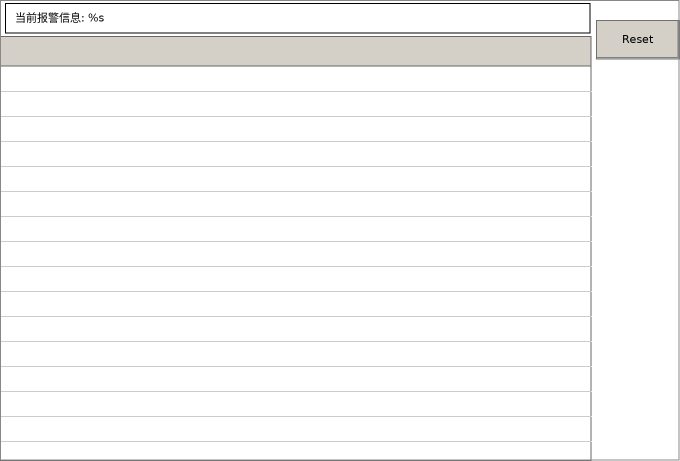
VISUALIZATION Visualization_ActEvent  // 680x461
    Button (596,20 84x39), "Reset"
        tap gvl.HMI_btReset
    Table (0,36 591x425), data array: AlarmActiveArray
        p3854506369: AlarmActiveArray[INDEX].EventMessage
        p1892666644: AlarmActiveArray[INDEX].EventId
        p338671338: AlarmActiveArray[INDEX].EventTime
    Rectangle (5,3 585x30), "当前报警信息: %s", text variable: gwsActEventMsg
END_VISUALIZATION

(* stored: Version 1.1.0.1, ProductVersion 3.1.4024.11
   Visu Visualization_ActEvent: Id {26cf3322-028f-491a-82c6-e4a2e718ba42} *)
